Staubli VAL3: setLoop.pgx

public program setLoop(bool x_bLoop)
  local string loop
begin
  // set the loop to ON OFF
  if x_bLoop
    loop="ON"
  else
    loop="OFF"
  endIf
  // set cycle LIST
  logMsg("[KERNEL] CYCLE:Set the loop mode to: "+loop)
  saveCycle:bLoop=x_bLoop
end
